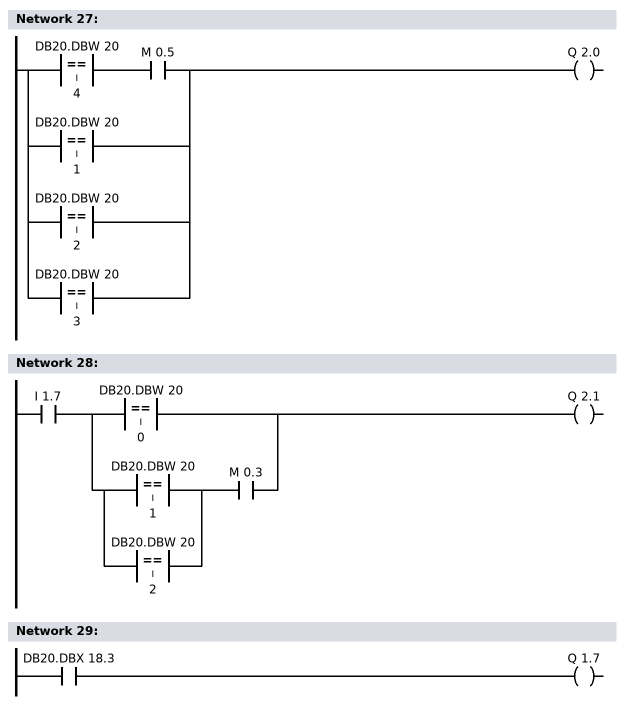
NETWORK
TITLE =
      A(;
      L     DB20.DBW 20;
      L     4;
      ==I;
      );
      A     M 0.5;
      O(;
      L     DB20.DBW 20;
      L     1;
      ==I;
      );
      O(;
      L     DB20.DBW 20;
      L     2;
      ==I;
      );
      O(;
      L     DB20.DBW 20;
      L     3;
      ==I;
      );
      =     Q 2.0;
NETWORK
TITLE =
      A     I 1.7;
      A(;
      O(;
      L     DB20.DBW 20;
      L     0;
      ==I;
      );
      O;
      A(;
      O(;
      L     DB20.DBW 20;
      L     1;
      ==I;
      );
      O(;
      L     DB20.DBW 20;
      L     2;
      ==I;
      );
      );
      A     M 0.3;
      );
      =     Q 2.1;
NETWORK
TITLE =
      A     DB20.DBX 18.3;
      =     Q 1.7;
END_FUNCTION_BLOCK

FUNCTION FC 1 : VOID
VERSION : 0.0
BEGIN
// body was compiled from an SCL source; compiled code not shown
END_FUNCTION

// FC 33: know-how protected block, not included

// FC 105: know-how protected block, not included

// FC 106: know-how protected block, not included

DATA_BLOCK DB 1
VERSION : 0.1
BEGIN
// 50 bytes; values not shown
END_DATA_BLOCK

DATA_BLOCK DB 2
VERSION : 0.1
BEGIN
// 22 bytes; values not shown
END_DATA_BLOCK

DATA_BLOCK DB 5
AUTHOR : SIMATIC
FAMILY : IEC_TC
VERSION : 0.0
SFB 4
BEGIN
END_DATA_BLOCK

DATA_BLOCK DB 6
AUTHOR : SIMATIC
FAMILY : IEC_TC
VERSION : 0.0
SFB 4
BEGIN
END_DATA_BLOCK

DATA_BLOCK DB 7
AUTHOR : SIMATIC
FAMILY : IEC_TC
VERSION : 0.0
SFB 4
BEGIN
END_DATA_BLOCK

DATA_BLOCK DB 8
AUTHOR : SIMATIC
FAMILY : IEC_TC
VERSION : 0.0
SFB 4
BEGIN
END_DATA_BLOCK

DATA_BLOCK DB 9
AUTHOR : SIMATIC
FAMILY : IEC_TC
VERSION : 0.0
SFB 4
BEGIN
END_DATA_BLOCK

DATA_BLOCK DB 10
AUTHOR : SIMATIC
FAMILY : IEC_TC
VERSION : 0.0
SFB 4
BEGIN
END_DATA_BLOCK

DATA_BLOCK DB 14
VERSION : 0.0
FB 3
BEGIN
END_DATA_BLOCK

DATA_BLOCK DB 15
VERSION : 0.0
FB 2
BEGIN
END_DATA_BLOCK

DATA_BLOCK DB 17
VERSION : 0.1
BEGIN
// 66 bytes; values not shown
END_DATA_BLOCK

DATA_BLOCK DB 18
VERSION : 0.1
BEGIN
// 66 bytes; values not shown
END_DATA_BLOCK

DATA_BLOCK DB 19
VERSION : 0.1
BEGIN
// 40 bytes; values not shown
END_DATA_BLOCK

DATA_BLOCK DB 20
VERSION : 0.1
BEGIN
// 38 bytes; values not shown
END_DATA_BLOCK

DATA_BLOCK DB 21
VERSION : 0.1
BEGIN
// 6 bytes; values not shown
END_DATA_BLOCK

DATA_BLOCK DB 22
VERSION : 0.1
BEGIN
// 6 bytes; values not shown
END_DATA_BLOCK

DATA_BLOCK DB 23
VERSION : 0.1
BEGIN
// 6 bytes; values not shown
END_DATA_BLOCK

DATA_BLOCK DB 24
VERSION : 0.1
BEGIN
// 6 bytes; values not shown
END_DATA_BLOCK

DATA_BLOCK DB 50
AUTHOR : SIMATIC
FAMILY : ICONT
VERSION : 0.0
FB 41
BEGIN
END_DATA_BLOCK

DATA_BLOCK DB 51
VERSION : 0.0
FB 50
BEGIN
END_DATA_BLOCK

DATA_BLOCK DB 52
VERSION : 0.0
FB 49
BEGIN
END_DATA_BLOCK

DATA_BLOCK DB 69
AUTHOR : SIMATIC
FAMILY : CONTROL
VERSION : 0.0
FB 58
BEGIN
END_DATA_BLOCK

DATA_BLOCK DB 70
AUTHOR : SIMATIC
FAMILY : CONTROL
VERSION : 0.0
FB 58
BEGIN
END_DATA_BLOCK

DATA_BLOCK DB 94
VERSION : 0.0
FB 94
BEGIN
END_DATA_BLOCK

DATA_BLOCK DB 95
VERSION : 0.0
FB 95
BEGIN
END_DATA_BLOCK

DATA_BLOCK DB 98
VERSION : 0.0
FB 98
BEGIN
END_DATA_BLOCK

DATA_BLOCK DB 99
VERSION : 0.0
FB 99
BEGIN
END_DATA_BLOCK

DATA_BLOCK DB 120
VERSION : 0.0
FB 20
BEGIN
END_DATA_BLOCK

DATA_BLOCK DB 130
AUTHOR : SIMATIC
FAMILY : CONTROL
VERSION : 0.0
FB 58
BEGIN
END_DATA_BLOCK

DATA_BLOCK DB 131
VERSION : 0.0
FB 47
BEGIN
END_DATA_BLOCK

DATA_BLOCK DB 132
VERSION : 0.0
FB 48
BEGIN
END_DATA_BLOCK

DATA_BLOCK DB 230
VERSION : 0.0
FB 20
BEGIN
END_DATA_BLOCK

DATA_BLOCK DB 231
AUTHOR : SIMATIC
FAMILY : CONTROL
VERSION : 0.0
FB 58
BEGIN
END_DATA_BLOCK

DATA_BLOCK DB 232
VERSION : 0.0
FB 5
BEGIN
END_DATA_BLOCK

ORGANIZATION_BLOCK OB 1
VERSION : 0.1
BEGIN
// (block stored without names or comments; labels and parameter names are numbered)
NETWORK
TITLE =
      UC    FB 1;
NETWORK
TITLE =
      CALL  FC 105 (
           $1                       := P#P 292.0,
           $2                       := L#1092616192,
           $3                       := L#0,
           $4                       := P#M 100.0,
           $5                       := DB1.DBW 36,
           $6                       := DB1.DBD 38);
      CALL  FC 105 (
           $1                       := P#P 294.0,
           $2                       := L#1092616192,
           $3                       := L#0,
           $4                       := P#M 100.0,
           $5                       := DB1.DBW 42,
           $6                       := DB1.DBD 44);
NETWORK
TITLE =
END_ORGANIZATION_BLOCK

ORGANIZATION_BLOCK OB 35
VERSION : 0.1
BEGIN
// (block stored without names or comments; labels and parameter names are numbered)
NETWORK
TITLE =
      CALL  FB 49 , DB 52;
      CALL  FB 50 , DB 51;
NETWORK
TITLE =
      CALL  FB 47 , DB 131;
      CALL  FB 48 , DB 132;
END_ORGANIZATION_BLOCK

ORGANIZATION_BLOCK OB 80
VERSION : 0.1
BEGIN
// (block stored without names or comments; labels and parameter names are numbered)
END_ORGANIZATION_BLOCK

ORGANIZATION_BLOCK OB 81
VERSION : 0.1
BEGIN
// (block stored without names or comments; labels and parameter names are numbered)
END_ORGANIZATION_BLOCK

ORGANIZATION_BLOCK OB 82
VERSION : 0.1
BEGIN
// (block stored without names or comments; labels and parameter names are numbered)
END_ORGANIZATION_BLOCK

ORGANIZATION_BLOCK OB 83
VERSION : 0.1
BEGIN
// (block stored without names or comments; labels and parameter names are numbered)
END_ORGANIZATION_BLOCK

ORGANIZATION_BLOCK OB 84
VERSION : 0.1
BEGIN
// (block stored without names or comments; labels and parameter names are numbered)
END_ORGANIZATION_BLOCK

ORGANIZATION_BLOCK OB 85
VERSION : 0.1
BEGIN
// (block stored without names or comments; labels and parameter names are numbered)
END_ORGANIZATION_BLOCK

ORGANIZATION_BLOCK OB 86
VERSION : 0.1
BEGIN
// (block stored without names or comments; labels and parameter names are numbered)
END_ORGANIZATION_BLOCK

ORGANIZATION_BLOCK OB 87
VERSION : 0.1
BEGIN
// (block stored without names or comments; labels and parameter names are numbered)
END_ORGANIZATION_BLOCK

ORGANIZATION_BLOCK OB 100
VERSION : 0.1
BEGIN
// (block stored without names or comments; labels and parameter names are numbered)
NETWORK
TITLE =
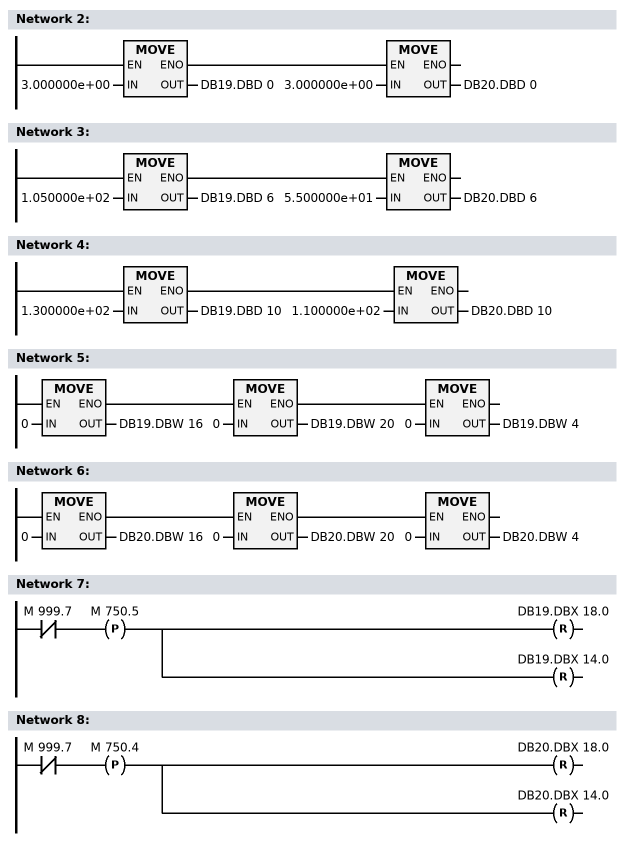
NETWORK
TITLE =
      A(;
      L     3.000000e+00;
      T     DB19.DBD 0;
      SET;
      SAVE;
      CLR;
      A     BR;
      );
      JNB   M001;
      L     3.000000e+00;
      T     DB20.DBD 0;
M001: NOP   0;
NETWORK
TITLE =
      A(;
      L     1.050000e+02;
      T     DB19.DBD 6;
      SET;
      SAVE;
      CLR;
      A     BR;
      );
      JNB   M002;
      L     5.500000e+01;
      T     DB20.DBD 6;
M002: NOP   0;
NETWORK
TITLE =
      A(;
      L     1.300000e+02;
      T     DB19.DBD 10;
      SET;
      SAVE;
      CLR;
      A     BR;
      );
      JNB   M003;
      L     1.100000e+02;
      T     DB20.DBD 10;
M003: NOP   0;
NETWORK
TITLE =
      A(;
      A(;
      L     0;
      T     DB19.DBW 16;
      SET;
      SAVE;
      CLR;
      A     BR;
      );
      JNB   M004;
      L     0;
      T     DB19.DBW 20;
      SET;
      SAVE;
      CLR;
M004: A     BR;
      );
      JNB   M005;
      L     0;
      T     DB19.DBW 4;
M005: NOP   0;
NETWORK
TITLE =
      A(;
      A(;
      L     0;
      T     DB20.DBW 16;
      SET;
      SAVE;
      CLR;
      A     BR;
      );
      JNB   M006;
      L     0;
      T     DB20.DBW 20;
      SET;
      SAVE;
      CLR;
M006: A     BR;
      );
      JNB   M007;
      L     0;
      T     DB20.DBW 4;
M007: NOP   0;
NETWORK
TITLE =
      AN    M 999.7;
      FP    M 750.5;
      R     DB19.DBX 18.0;
      R     DB19.DBX 14.0;
NETWORK
TITLE =
      AN    M 999.7;
      FP    M 750.4;
      R     DB20.DBX 18.0;
      R     DB20.DBX 14.0;
END_ORGANIZATION_BLOCK

ORGANIZATION_BLOCK OB 101
VERSION : 0.1
BEGIN
// (block stored without names or comments; labels and parameter names are numbered)
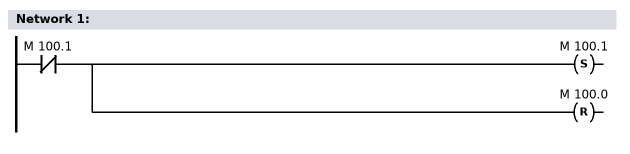
NETWORK
TITLE =
      AN    M 100.1;
      S     M 100.1;
      R     M 100.0;
END_ORGANIZATION_BLOCK

ORGANIZATION_BLOCK OB 102
VERSION : 0.1
BEGIN
// (block stored without names or comments; labels and parameter names are numbered)
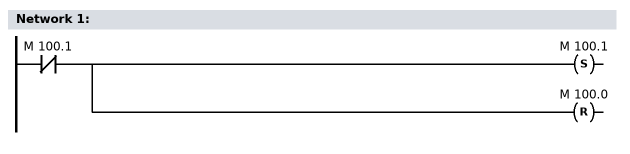
NETWORK
TITLE =
      AN    M 100.1;
      S     M 100.1;
      R     M 100.0;
END_ORGANIZATION_BLOCK

ORGANIZATION_BLOCK OB 121
VERSION : 0.1
BEGIN
// (block stored without names or comments; labels and parameter names are numbered)
END_ORGANIZATION_BLOCK
